// TIA Portal V20 export
DATA_BLOCK "Config"   // DB106
// stored: Access Published, MemoryReserve 100, Namespace Unit1.Em6
   VAR
      em : "LAF_typeEmConfiguration";   // Configuration of EM Parameters
      axis : Array[1.._.U1EM6_NO_OF_AXES] of DB_ANY;
      cam : Array[1.._.U1EM6_NO_OF_AXES] of DB_ANY;
      outputCam : Array[1.._.U1EM6_NO_OF_AXES] of DB_ANY;
      moduleAccessPoint : Array[1.._.U1EM6_NO_OF_AXES] of HW_SUBMODULE;
   END_VAR
   VAR RETAIN
      cmVisionUnitAxisZ : "LBC_typeAxis64PosConfiguration";
      cmVisionPusherSupportUpDown : "LBC_typeTwoWayActuatorConfiguration";
      cmVisionTriggerSensor : "LBC_typeDigitalSignalConfiguration";
      cmVisionController : "LER_typeVisionConfiguration";
      cmQrReader : "LER_typeSRX300Configuration";
      cmQrReaderHandy : "LER_typeDM8700Configuration";
      cmVisionUnitAxisZ_TorqueCal : "LER_typeServoTorqueCalConfigruation";
   END_VAR
BEGIN
   // axis[1] : cmVisionUnitAxisZ
   // cam[1] : cmVisionUnitAxisZ
   // moduleAccessPoint[1] : cmVisionUnitAxisZ
   cmQrReader.hwID.handshakeGeneralErrorStatusHwId := 538;
   cmQrReader.hwID.busyStatusHwId := 537;
   cmQrReader.hwID.completionStatusHwId := 536;
   cmQrReader.hwID.errorStatusHwId := 535;
   cmQrReader.hwID.terminalStatusHwId := 534;
   cmQrReader.hwID.unstableReadStatusHwId := 533;
   cmQrReader.hwID.matchingAndGradeStatusHwId := 532;
   cmQrReader.hwID.operationResultStatusHwId := 531;
   cmQrReader.hwID.readDataHeaderHwId := 530;
   cmQrReader.hwID.readDataExtendedPart1HwId := 530;
   cmQrReader.hwID.readDataExtendedPart2HwId := 530;
   cmQrReader.hwID.readDataExtendedPart3HwId := 530;
   cmQrReader.hwID.latchErrorClearControlHwId := 529;
   cmQrReader.hwID.operationInstructionControlHwId := 528;
   cmQrReader.hwID.completionClearControlHwId := 484;
   cmQrReader.hwID.parameterBankNumberHwId := 483;
   cmQrReader.hwID.userDataHwId := 482;
   cmQrReaderHandy.hwID.Acquisition_Status_HW_ID := 1;
   cmQrReaderHandy.hwID.Results_Status_HW_ID := 1;
   cmQrReaderHandy.hwID.Soft_Event_Status_HW_ID := 1;
   cmQrReaderHandy.hwID.Result_Data_HW_ID := 1;
   cmQrReaderHandy.hwID.Acquisition_Control_HW_ID := 1;
   cmQrReaderHandy.hwID.Results_Control_HW_ID := 1;
   cmQrReaderHandy.hwID.Soft_Event_Control_HW_ID := 1;
   cmQrReaderHandy.hwID.User_Data_HW_ID := 1;
   cmQrReaderHandy.disableAlarms := True;
END_DATA_BLOCK
